RoboDK station: Clase1IndustrialRobotics.rdk

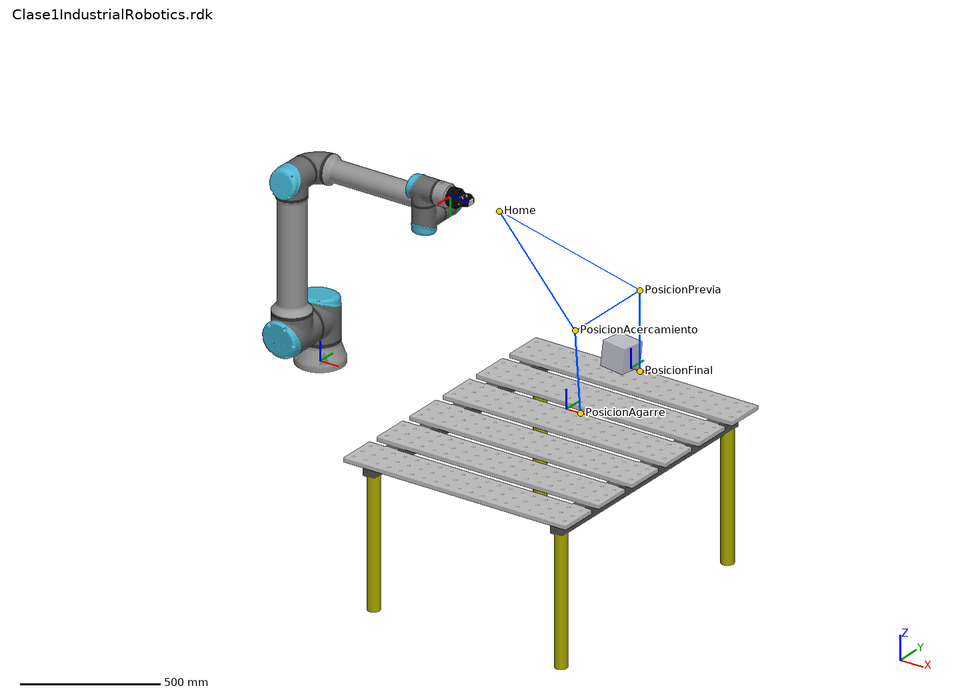
[picture v0: the station drawn from its stored meshes, robots at their saved joint values, targets as dots, program paths as lines]
Station Clase1IndustrialRobotics (saved by RoboDK 5.5.0). Poses are relative to the parent item; angles as X-Y-Z fixed-axis rotations.
  - frame UR10e Base at (0, 0, 0) mm
    - robot UR10e: 6 axes, payload 10 kg, reach 1300 mm, repeatability 0.05 mm, weight 28.9 kg
        modified DH rows (alpha deg, a mm, theta deg, d mm): 0, 0, 0, 180.7; 90, 0, 180, 0; 0, 612.6, 0, 0; 0, 571.335, 0, 174.15; -90, 0, 0, 119.85; 90, 0, 180, 116.55
        joint limits [-360, -360, -360, -360, -360, -360] to [360, 360, 360, 360, 360, 360]; home [0, -90, -90, 0, 90, 0]; saved at [0, -90, -90, 0, 90, 0]
      - frame RobotiQ 2F85 Base at (0, 0, 0) mm
        - robot RobotiQ 2F85: 1 axes, payload 5 kg
            joint limits [0] to [85]; home [85]; saved at [85]
        - target Open (Cartesian target) at (938.55, 100, 246.18) mm, rotated rx -85.99 ry 0 rz -90 deg; joints [85] of RobotiQ 2F85
        - target Close (Cartesian target) at (0, 0, 103.92) mm; joints [68.98] of RobotiQ 2F85
      - tool 2F85, TCP at (0, 0, 211.5) mm
    - target PosicionAgarre (Cartesian target) at (1059.85, 100, 50) mm, rotated rx -85.99 ry 0 rz -90 deg; joints [21.396, -153.863, -98.022, 76.192, 68.659, -1.57] of UR10e
    - target Home (Cartesian target) at (899.38, -174.15, 913.15) mm, rotated rx -90 ry 0 rz -90 deg; joints [0, -90, -90, 0, 90, 0] of UR10e
    - target PosicionAcercamiento (Cartesian target) at (1037.47, 100, 369.22) mm, rotated rx -85.99 ry 0 rz -90 deg; joints [22.067, -125.528, -106.843, 56.698, 67.99, -1.624] of UR10e
    - target PosicionPrevia (Cartesian target) at (1037.47, 500, 369.22) mm, rotated rx -85.99 ry 0 rz -90 deg; joints [46.712, -135.658, -86.279, 47.776, 43.437, -4.247] of UR10e
    - target PosicionFinal (Cartesian target) at (1037.47, 500, 50) mm, rotated rx -85.99 ry 0 rz -90 deg; joints [46.712, -159.071, -80.316, 65.226, 43.437, -4.247] of UR10e
  - object Table at (1000, 0, 0) mm, rotated rx 0 ry 0 rz 90 deg, size 1193.8 x 965.2 x 609.6 mm, geometry from welding_table.sld
  - frame PosicionA at (1000, 100, 50) mm
  - frame PosicionB at (1000, 500, 50) mm
    - object box at (-40.58, -3.89, 50) mm, rotated rx -4.01 ry 3.72 rz -4.28 deg, size 100 x 100 x 100 mm, geometry from box.sld
  - program ProgramaPrincipal (14 instructions, listed below)
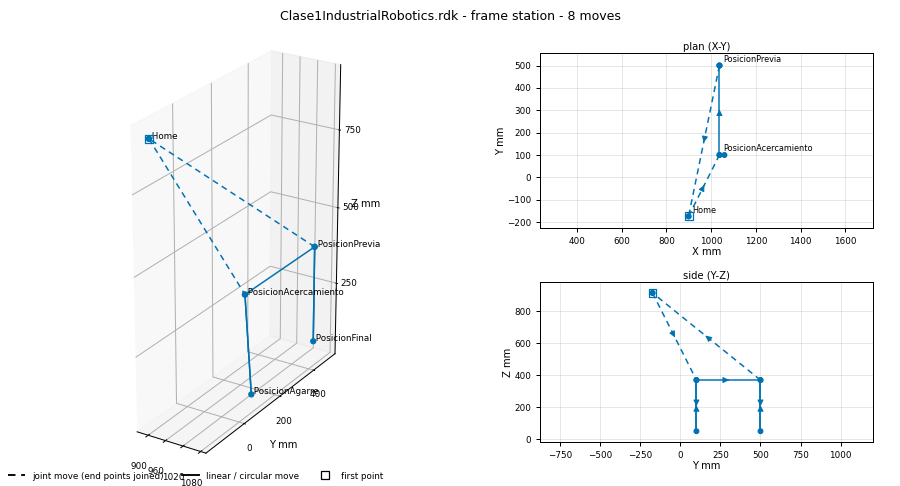
[picture p0: tool path of Clase1IndustrialRobotics.rdk in frame station, 8 of 8 moves have a stored position in this frame; points joined in program order, loops and branches not executed]

--- program ProgramaPrincipal (robot UR10e) ---
  Est. Ref.: UR10e Base
  Est. herr: 2F85
  MoveJ (Home)
  MoveJ (PosicionAcercamiento)
  MoveL (PosicionAgarre)
  Adjuntar a 2F85
  MoveL (PosicionAcercamiento)
  Establecer velocidad (50.0 mm/s)
  MoveL (PosicionPrevia)
  MoveL (PosicionFinal)
  Separar de 2F85
  MoveL (PosicionPrevia)
  Establecer velocidad (500.0 mm/s)
  MoveJ (Home)
